// TIA Portal V20 export
DATA_BLOCK "ControlNodes"   // DB164
// stored: MemoryReserve 100, Namespace Unit1.Em1
   VAR
      em { ExternalWritable := 'False'} : "LAF_typeEmControlNode";
      emstate { S7_SetPoint := 'True'} : "LUC_typeStates";
      cm : "Unit1.Em1.typeCmControlNode";
      citiMap : Struct
         PMC : "LER_PMC_Input_Data";
         FlexNet { S7_SetPoint := 'True'} : "LER_FlexNet_Data";
      END_STRUCT;
      stacker2NgBox : "Unit1.Em1.typeSequenceControlNode";
      SpecialFunctionMode : Struct
         DryRun : Struct
            JRdetectPV : Array[0..15] of Bool;
         END_STRUCT;
      END_STRUCT;
      unitCommunication : "Unit1.Em1.typeUnitCommunicationControlNode";
      cmStacker2NgBoxDetect { S7_SetPoint := 'True'} : "LBC_typeDigitalSignalControlNode";
      cmStacker2NgBoxFullDetect { S7_SetPoint := 'True'} : "LBC_typeDigitalSignalControlNode";
      cmStacker2NgBoxLoadingUpDown { S7_SetPoint := 'True'} : "LBC_typeTwoWayActuatorControlNode";
      cmStacker2NgBoxUnitMoverBwdFwd { S7_SetPoint := 'True'} : "LBC_typeTwoWayActuatorControlNode";
      cmStacker2NgBoxClampLeftOpenClose { S7_SetPoint := 'True'} : "LBC_typeTwoWayActuatorControlNode";
      cmStacker2NgBoxClampRightOpenClose { S7_SetPoint := 'True'} : "LBC_typeTwoWayActuatorControlNode";
      cmStacker2NgBoxClampMoverOpenClose { S7_SetPoint := 'True'} : "LBC_typeTwoWayActuatorControlNode";
      cmStacker2NgBoxLiftDownUp { S7_SetPoint := 'True'} : "LBC_typeTwoWayActuatorControlNode";
      cmStacker2NgBoxLockDownUp { S7_SetPoint := 'True'} : "LBC_typeTwoWayActuatorControlNode";
   END_VAR
BEGIN
END_DATA_BLOCK
